PROGRAM MAIN
VAR
END_VAR

END_PROGRAM

(* stored: Version 1.1.0.1
   POU MAIN: Id {40a4b2da-b081-4022-8cc5-935887cb0bb9} *)
